FUNCTION_BLOCK FB_BaseMotor IMPLEMENTS I_Motor

VAR
	nMotorSpeed : INT;
	bEnable : BOOL;
END_VAR

{warning 'add method implementation '}
METHOD DrySpin : BOOL
VAR_INPUT
	nMotorSpeed	: INT;
END_VAR
END_METHOD

{warning 'add method implementation '}
METHOD ForwardSpin : BOOL
VAR_INPUT
	nMotorSpeed	: INT;
END_VAR
bEnable := TRUE;
END_METHOD

METHOD Stop : BOOL
VAR_INPUT
END_VAR
bEnable := FALSE;
END_METHOD

END_FUNCTION_BLOCK

(* stored: Version 1.1.0.1, ProductVersion 3.1.4024.16
   POU FB_BaseMotor: Id {fc772ccd-6811-433f-bdff-1beb293d4214}, SpecialFunc None
   Method DrySpin: Id {ef8e60bc-43e2-4077-a193-f1d492cbfc42}
   Method ForwardSpin: Id {e526ef12-d8c4-41df-8d3e-ca783664064a}
   Method Stop: Id {6ac747cd-6170-4826-8baa-995ada24ee4f} *)
